Fanuc KAREL source: CNV_REL_JPOS.kl

PROGRAM T
%NOLOCKGROUP
VAR
 v0 : ARRAY[9] OF REAL
 v1 : JOINTPOS
 v2 : INTEGER
BEGIN
 CNV_REL_JPOS(v0, v1, v2)
END T
